FUNCTION_BLOCK TrueUntil (* Basic Function Block Type *)
  (* Standard: 61499-2 *)
  (* Version 0.0, 2/9/2018, Sandeep Patil, nxtControl GmbH, Template *)
  PACKAGE Main;
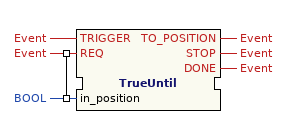
  EVENT_INPUT
    TRIGGER; (* Initialization Request *)
    REQ WITH in_position; (* Normal Execution Request *)
  END_EVENT
  EVENT_OUTPUT
    TO_POSITION; (* Initialization Confirm *)
    STOP; (* Execution Confirmation *)
    DONE;
  END_EVENT
  VAR_INPUT
    in_position : BOOL;
  END_VAR
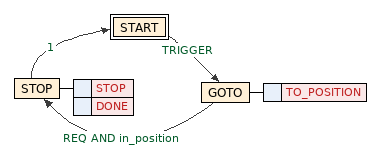
  EC_STATES
    START; (* Initial State *)
    STOP : -> STOP, -> DONE;
    GOTO : -> TO_POSITION;
  END_STATES
  EC_TRANSITIONS
    GOTO TO STOP := REQ AND in_position;
    STOP TO START := 1;
    START TO GOTO := TRIGGER;
  END_TRANSITIONS
  ALGORITHM INIT IN ST: (* Initialization algorithm *)
;
  END_ALGORITHM
  ALGORITHM REQ IN ST: (* Normally executed algorithm *)
;
  END_ALGORITHM
END_FUNCTION_BLOCK
